PROGRAM prg_Click_Log
VAR
END_VAR

END_PROGRAM

(* stored: Version 1.1.0.1, ProductVersion 3.1.4024.15
   POU prg_Click_Log: Id {bdf18c93-f4bb-492e-a5f7-46873c367823}, SpecialFunc None *)
